PROGRAM MAIN_10MS
VAR
END_VAR

// NETWORK 1

END_PROGRAM

(* stored: Version 1.1.0.1, ProductVersion 3.1.4024.12
   POU MAIN_10MS: Id {72a9e298-3ada-4b58-83f7-1604d2f7bd42}, SpecialFunc None *)
